{attribute 'GeneratedUsingTerminal: ER4374-0002-0018'}
{attribute addProperty BoxType "ER4374-0002-0018"}
{attribute addProperty Id "StatusAT %I*Status_B07533568ValueAT %I*INT2"}
{attribute addProperty CRC "2833212643"}
{attribute addProperty Size "10"}
TYPE AI_Inputs_Channel_A8DF64E3 :
STRUCT
	{attribute addProperty Name "Status"}
	Status AT %I* : Status_B0753356;
	{attribute addProperty Name "Value"}
	Value AT %I* : INT;
END_STRUCT
END_TYPE

(* stored: Version 1.2.0.0, ProductVersion 3.1.4024.9
   DUT AI_Inputs_Channel_A8DF64E3: Id {a59fe3fc-01ef-43c4-801e-5d798d4c3a0c} *)
